// TwinCAT 3 PLC project Plc
// ProgramVersion: 3.1.4024.0
// libraries:
//   Tc2_Math, * (Beckhoff Automation GmbH)
//   Tc2_MC2, * (Beckhoff Automation GmbH)
//   Tc2_Standard, * (Beckhoff Automation GmbH)
//   Tc2_System, * (Beckhoff Automation GmbH)
//   Tc3_Module, * (Beckhoff Automation GmbH)
// project tree:
//   DUTs/ E_Aquisition_State.TcDUT, E_TestAccuracy_State.TcDUT
//   GVLs/ GVL_AccuracyTest.TcGVL, GVL_Interpolation.TcGVL
//   / PlcTask.TcTTO
//   POUs/ Accuracy_Measurement.TcPOU, MAIN.TcPOU, PositionCompensation_1D.TcPOU
//   POUs/Maths/ average.TcPOU, max_abs_array.TcPOU, max_array.TcPOU, min_array.TcPOU, scaling.TcPOU, sigma.TcPOU
// real-time tasks:
//   TASK Task_Plc: cycle T#2ms, priority 20, ADS port 350
// motion (NC):
//   TASK NC-Task 1 SAF: cycle T#2ms, priority 4, ADS port 501
//   TASK NC-Task 1 SVB: cycle T#10ms, priority 8, ADS port 511
//   AXIS Axis 1 (id 1)
//     Dynamic: Acceleration=1225.67, Deceleration=1225.67, Jerk=3677.02
//     Velo: RefSearch=8.17116, RefSync=8.17116, SlowManual=40.8558, FastManual=245.1348, Fast=817.116, Maximum=817.116
//     TargetPosControl: Range=0.0002, Time=0.1
//     OtherSettings: AllowMotionCmdToSlave=true
//     encoder EncType=19
//       EncPara: ScaleFactorNumerator=10, ScaleFactorDenominator=1048576, MaxCount=#xffffffff
//         SoftEndMinControl: Enable=true, Range=-170
//         SoftEndMaxControl: Enable=true, Range=30
//     drive DrvType=16
//       DrvPara: MaxCount=#xffffffff, DriveControlDWord=#x00020100
//         Analog: VeloReferenz=898.8276, VeloScale=71.5255737304688, TorqueSetpointScale=10, ScaleFactorActTorque=0.1
//         TimeComp: TaskDelayCycles=1
//     controller CtrType=1
//       CtrPara: PriorControlFactor=1
//         Observer: BandWidth=20
//   AXIS Axis 2 (id 2)
//     Dynamic: Acceleration=5539.8765, Deceleration=5539.8765, Jerk=16619.6295
//     Velo: RefSearch=36.93251, RefSync=36.93251, SlowManual=184.66255, FastManual=1107.9753, Fast=3693.251, Maximum=3693.251
//     TargetPosControl: Range=0.0005, Time=0.1
//     OtherSettings: AllowMotionCmdToSlave=true
//     encoder EncType=19
//       EncPara: ScaleFactorNumerator=60, ScaleFactorDenominator=1048576, MaxCount=#xffffffff
//     drive DrvType=16
//       DrvPara: MaxCount=#xffffffff, DriveControlDWord=#x00020100
//         Analog: VeloReferenz=4062.5761, VeloScale=71.5255737304688, TorqueSetpointScale=10, ScaleFactorActTorque=0.1
//         TimeComp: TaskDelayCycles=1
//     controller CtrType=1
//       CtrPara: PriorControlFactor=1
//         Observer: BandWidth=20
// I/O:
//   DEVICE Device 1 (EtherCAT) (disabled), AmsNetId 5.64.37.70.2.1
//     Term 1 (EK1200) [EK1200-5000 EtherCAT Power supply (2A E-Bus)]
//       Term 2 (EL6910) [EL6910, TwinSAFE PLC]
//       Term 3 (EL1904) [EL1904, 4 Ch. Safety Input 24V, TwinSAFE]
//         modules: Module 1 (FSOES)
//       Term 4 (EL1008) [EL1008 8Ch. Dig. Input 24V, 3ms]
//       Term 5 (EL9011) [EL9011 End Terminal]
//   DEVICE Device 4 (EtherCAT), AmsNetId 5.64.37.70.5.1
//     Term 6 (AX8620-0000-0103) [AX8620-0000-0103]
//       Drive 7 (AX8206-0210-0106) [AX8206-0210-0106 (2Ch. 6A servo axis, safe-motion, multi-FB)]
//         modules: Device, Device, Device, Device, Device, Device, Device, Device, Device, Device, Device (Safety), Device, Device, Device, Device, Device, Device, Device, Device, Device, Device, Device, Device, Device, Device, Device, Device, Device, Device, Device, Device, Ch A, Ch A, Ch A, Ch A, Ch A, Ch A, Ch A, Ch A, Ch A, Ch A, Ch A, Ch A, Ch A, Ch A, Ch A, Ch A, Ch A, Ch A, Ch A, Ch A, Ch A, Ch A, Ch A, Ch A, Ch A, Ch A, Ch A, Ch B, Ch B, Ch B, Ch B, Ch B, Ch B, Ch B, Ch B, Ch B, Ch B, Ch B, Ch B, Ch B, Ch B, Ch B, Ch B, Ch B, Ch B, Ch B, Ch B, Ch B, Ch B, Ch B, Ch B, Ch B, Ch B
//         startup 12992:1 := 414D383032312D78427830 // Ch A Motor parameters / Configured motor type
//         startup 24768:0 := FEFF // Ch A Interpolation sub mode select
//         startup 13000:5 := 0200 // Ch A Motor thermal model / Reaction
//         startup 13000:6 := 0000C841 // Ch A Motor thermal model / Partial fraction factor
//         startup 12992:12 := 0000FA45 // Ch A Motor parameters / Motor rated speed
//         startup 12992:13 := C9E5FF3E // Ch A Motor parameters / Motor rated torque
//         startup 24694:0 := F4010000 // Ch A Motor standstill torque
//         startup 24800:0 := D007 // Ch A Positive torque/force limit value
//         startup 24801:0 := D007 // Ch A Negative torque/force limit value
//         startup 12288:6 := 4158383230362D303231302D30303030 // Ch A AxisMain parameters / Configured drive type
//         startup 12867:1 := 9A99593F // Ch A TorqueCtrl parameters / Configured channel rated current
//         startup 12867:2 := 33332340 // Ch A TorqueCtrl parameters / Configured channel peak current
//         startup 12867:7 := 77BE1F40 // Ch A TorqueCtrl parameters / Iuvw max sum
//         startup 24672:0 := 08 // Ch A Modes of operation
//         startup 13023:0 := 0000 // Ch A Motor control mode
//         startup 12864:1 := 0D4D7043 // Ch A TorqueCtrl parameters mappable / Torque control proportional gain q
//         startup 12864:2 := 8A0E7C39 // Ch A TorqueCtrl parameters mappable / Torque control integral action time q
//         startup 12608:1 := FBD1CD3B // Ch A VeloCtrl parameters mappable / Velocity control proportional gain
//         startup 12608:2 := 6F12033C // Ch A VeloCtrl parameters mappable / Velocity control integral action time
//         startup 12608:3 := 00980546 // Ch A VeloCtrl parameters mappable / Bipolar velocity limit value
//         startup 12992:15 := 0100 // Ch A Motor parameters / Motor temperature sensor connection
//         startup 12611:4 := 0400 // Ch A VeloCtrl observer / Observer type
//         startup 24672:0 := 08 // Ch A Modes of operation
//         startup 12296:2 := 00 // Ch A AxisMain parameters encoder direction / Primary encoder direction
//         startup 12296:1 := 00 // Ch A AxisMain parameters encoder direction / Secondary encoder direction
//         startup 14016:1 := 414D383033332D78467831 // Ch B Motor parameters / Configured motor type
//         startup 26816:0 := FEFF // Ch B Interpolation sub mode select
//         startup 14024:5 := 0200 // Ch B Motor thermal model / Reaction
//         startup 14024:6 := 0000C841 // Ch B Motor thermal model / Partial fraction factor
//         startup 14016:12 := 0080BB45 // Ch B Motor parameters / Motor rated speed
//         startup 14016:13 := 2FDD3440 // Ch B Motor parameters / Motor rated torque
//         startup 26742:0 := 920C0000 // Ch B Motor standstill torque
//         startup 26848:0 := D007 // Ch B Positive torque/force limit value
//         startup 26849:0 := D007 // Ch B Negative torque/force limit value
//         startup 13312:6 := 4158383230362D303231302D30303030 // Ch B AxisMain parameters / Configured drive type
//         startup 13891:1 := 33338340 // Ch B TorqueCtrl parameters / Configured channel rated current
//         startup 13891:2 := CDCC4441 // Ch B TorqueCtrl parameters / Configured channel peak current
//         startup 13891:7 := 77BE1F40 // Ch B TorqueCtrl parameters / Iuvw max sum
//         startup 26720:0 := 08 // Ch B Modes of operation
//         startup 14047:0 := 0000 // Ch B Motor control mode
//         startup 13888:1 := 3DD94842 // Ch B TorqueCtrl parameters mappable / Torque control proportional gain q
//         startup 13888:2 := 8A0E7C39 // Ch B TorqueCtrl parameters mappable / Torque control integral action time q
//         startup 13632:1 := 4D288C3D // Ch B VeloCtrl parameters mappable / Velocity control proportional gain
//         startup 13632:2 := 6F12033C // Ch B VeloCtrl parameters mappable / Velocity control integral action time
//         startup 13632:3 := 00980546 // Ch B VeloCtrl parameters mappable / Bipolar velocity limit value
//         startup 14016:15 := 0100 // Ch B Motor parameters / Motor temperature sensor connection
//         startup 13635:4 := 0400 // Ch B VeloCtrl observer / Observer type
//         startup 26720:0 := 08 // Ch B Modes of operation
//         startup 13320:2 := 00 // Ch B AxisMain parameters encoder direction / Primary encoder direction
// variable links:
//   Device 4 (EtherCAT) <-> Device 4 (EtherCAT)/Term 6 (AX8620-0000-0103)/Drive 7 (AX8206-0210-0106)
//     Term 6 (AX8620-0000-0103)/PSM Controlword for axis/Controlword for axis <-> Device/DeviceMain Outputs/Power supply controlword
//   NC-Task 1 SAF/Axes/Axis 1 <-> Device 4 (EtherCAT)/Term 6 (AX8620-0000-0103)/Drive 7 (AX8206-0210-0106)
//     Drive/Inputs/In/nDataIn1 <-> Ch A/Ch A PositionControl Inputs/Ch A Following error actual value
//     Drive/Inputs/In/nDataIn3[0] <-> Ch A/Ch A TorqueControl Inputs/Ch A Torque/force actual value
//     Drive/Inputs/In/nDcOutputTime <-> InfoData/DcOutputShift
//     Drive/Inputs/In/nState1 <-> Ch A/Ch A AxisMain Inputs/Ch A Statusword
//     Drive/Inputs/In/nState2 <-> Ch A/Ch A AxisMain Inputs/Ch A Statusword @bit 8
//     Drive/Inputs/In/nState4 @bit 1 <-> WcState/InputToggle0
//     Drive/Inputs/In/nState4 <-> WcState/WcState0
//     Drive/Outputs/Out/nCtrl1 <-> Ch A/Ch A AxisMain Outputs/Ch A Controlword
//     Drive/Outputs/Out/nCtrl2 <-> Ch A/Ch A AxisMain Outputs/Ch A Controlword @bit 8
//     Drive/Outputs/Out/nDataOut1 <-> Ch A/Ch A Interpolator Outputs/Ch A Target position
//     Drive/Outputs/Out/nDataOut2 <-> Ch A/Ch A Interpolator Outputs/Ch A Target velocity
//     Enc/Inputs/In/nDataIn1 <-> Ch A/Ch A AxisMain Inputs/Ch A Position actual value
//     Enc/Inputs/In/nDcInputTime <-> InfoData/DcInputShift
//     Enc/Inputs/In/nState2 @bit 5 <-> Ch A/Ch A AxisMain Inputs/Position actual value invalid
//     Enc/Inputs/In/nState4 @bit 1 <-> WcState/InputToggle0
//     Enc/Inputs/In/nState4 <-> WcState/WcState0
//   NC-Task 1 SAF/Axes/Axis 2 <-> Device 4 (EtherCAT)/Term 6 (AX8620-0000-0103)/Drive 7 (AX8206-0210-0106)
//     Drive/Inputs/In/nDataIn1 <-> Ch B/Ch B PositionControl Inputs/Ch B Following error actual value
//     Drive/Inputs/In/nDcOutputTime <-> InfoData/DcOutputShift
//     Drive/Inputs/In/nState1 <-> Ch B/Ch B AxisMain Inputs/Ch B Statusword
//     Drive/Inputs/In/nState2 <-> Ch B/Ch B AxisMain Inputs/Ch B Statusword @bit 8
//     Drive/Inputs/In/nState4 @bit 1 <-> WcState/InputToggle0
//     Drive/Inputs/In/nState4 <-> WcState/WcState0
//     Drive/Outputs/Out/nCtrl1 <-> Ch B/Ch B AxisMain Outputs/Ch B Controlword
//     Drive/Outputs/Out/nCtrl2 <-> Ch B/Ch B AxisMain Outputs/Ch B Controlword @bit 8
//     Drive/Outputs/Out/nDataOut1 <-> Ch B/Ch B Interpolator Outputs/Ch B Target position
//     Drive/Outputs/Out/nDataOut2 <-> Ch B/Ch B Interpolator Outputs/Ch B Target velocity
//     Enc/Inputs/In/nDataIn1 <-> Ch B/Ch B AxisMain Inputs/Ch B Position actual value
//     Enc/Inputs/In/nDcInputTime <-> InfoData/DcInputShift
//     Enc/Inputs/In/nState2 @bit 5 <-> Ch B/Ch B AxisMain Inputs/Position actual value invalid
//     Enc/Inputs/In/nState4 @bit 1 <-> WcState/InputToggle0
//     Enc/Inputs/In/nState4 <-> WcState/WcState0
//   Plc/Plc Instance <-> Device 4 (EtherCAT)/Term 6 (AX8620-0000-0103)/Drive 7 (AX8206-0210-0106)
//     PlcTask Inputs/Accuracy_Measurement.iLastPositionRaw <-> Ch A/Ch A AxisMain Inputs/1st additional position actual value
//   Plc/Plc Instance <-> NC-Task 1 SAF/Axes/Axis 1
//     PlcTask Inputs/Accuracy_Measurement.Axis.NcToPlc <-> Outputs/ToPlc
//     PlcTask Outputs/Accuracy_Measurement.Axis.PlcToNc <-> Inputs/FromPlc

CONFIGURATION Plc
    RESOURCE PLC ON TwinCAT3
        TASK PlcTask(INTERVAL := T#2ms, PRIORITY := 20);
        PROGRAM MAIN WITH PlcTask : MAIN;
    END_RESOURCE
END_CONFIGURATION

// ---- DUTs/E_Aquisition_State.TcDUT
{attribute 'qualified_only'}
{attribute 'strict'}
TYPE E_Aquisition_State :
(
	IDLE := 0,
	MOVE_TO_FIRST_POS,
	WAIT_MOVE_TO_FIRST_POS,
	MOVE_TO_TARGET_FORWARD,
	WAIT_MOVE_TO_TARGET_FORWARD,
	MOVE_TO_LAST_POS,
	WAIT_MOVE_TO_LAST_POS,
	MOVE_TO_TARGET_BACKWARD,
	WAIT_MOVE_TO_TARGET_BACKWARD,
	DONE
);
END_TYPE

// ---- DUTs/E_TestAccuracy_State.TcDUT
{attribute 'qualified_only'}
{attribute 'strict'}
TYPE E_TestAccuracy_State :
(
	IDLE := 0,
	MOVE_TO_FIRST_POS,
	WAIT_MOVE_TO_FIRST_POS,
	MOVE_TO_TARGET_FORWARD,
	WAIT_MOVE_TO_TARGET_FORWARD,
	MOVE_TO_LAST_POS,
	WAIT_MOVE_TO_LAST_POS,
	MOVE_TO_TARGET_BACKWARD,
	WAIT_MOVE_TO_TARGET_BACKWARD,
	DONE
);
END_TYPE

// ---- GVLs/GVL_AccuracyTest.TcGVL
{attribute 'qualified_only'}
VAR_GLOBAL CONSTANT
	N_NBR_POSITIONS 	: UINT := 10;
	N_NBR_CYCLES 		: UINT := 5;
	N_NBR_DELAY_CYCLES 	: UINT := 5;
END_VAR

// ---- GVLs/GVL_Interpolation.TcGVL
{attribute 'qualified_only'}
VAR_GLOBAL
	N_MAX_POINTS : UINT := 10;
END_VAR

// ---- POUs/MAIN.TcPOU
PROGRAM MAIN
VAR 
END_VAR

Accuracy_Measurement();

END_PROGRAM

// ---- POUs/Accuracy_Measurement.TcPOU
PROGRAM Accuracy_Measurement
VAR
	
{region 'Axis Control FB'}	
	fbAxis 						: AXIS_REF;			// Axis to be moved
	
	fbPower						: MC_Power;			// Power the axis
	bPower						: BOOL;
	                			
	fbMove						: MC_MoveAbsolute;  // Move the axis
	bMove						: BOOL;
	fTarget						: LREAL;
	fVelocity					: LREAL := 100;
	fAcceleration				: LREAL;
	fJerk 						: LREAL;
	stOutputs					: ST_McOutputs;
		 
	fPositionError				: LREAL;			// Load Following error
	aRollingBuffer				: ARRAY[1..GVL_AccuracyTest.N_NBR_DELAY_CYCLES] OF LREAL; // Dead time of set pos
		 
	
	fbCompensation				: PositionCompensation_1D;  // Compensation
{endregion}	      	
	 
{region 'Load Position'}
	nLoadPositionRaw AT%I*		: DINT;				// Raw 
	fLoadPositionScaled 		: LREAL;			// Scaled Position in NC unit
	fLoadPositionOffset 		: LREAL := -74.157595; // To be calibrated for the current axis
{endregion}	

{region 'Cycle control'}	
	aSetposition				: ARRAY[1..GVL_AccuracyTest.N_NBR_POSITIONS] OF LREAL; // all positions for the measurement
	aMeasuredData				: ARRAY[1..GVL_AccuracyTest.N_NBR_POSITIONS, 1..2*GVL_AccuracyTest.ciNumCycles] OF LREAL; // Cycles : odd = forward, even = backward
	nCurrentSetpoint 			: UINT;			//
	nCurrentCycle	  			: UINT;
	bBackward					: BOOL;		     // Moving Backward
	fPositionMin				: LREAL := -170; // initialized from the NC
	fPositionMax				: LREAL := 30;   // initialized from the NC
	fStep						: LREAL;
{endregion}

{region 'ISO 230-2 metrics'}	
	aAverageForward					: ARRAY[1..GVL_AccuracyTest.N_NBR_POSITIONS] OF LREAL; 
	aAverageBackward				: ARRAY[1..GVL_AccuracyTest.N_NBR_POSITIONS] OF LREAL; 
	aAverageBidir					: ARRAY[1..GVL_AccuracyTest.N_NBR_POSITIONS] OF LREAL; 
	aSigmaForward					: ARRAY[1..GVL_AccuracyTest.N_NBR_POSITIONS] OF LREAL; 
	aSigmaBackward					: ARRAY[1..GVL_AccuracyTest.N_NBR_POSITIONS] OF LREAL; 
	aReversal						: ARRAY[1..GVL_AccuracyTest.N_NBR_POSITIONS] OF LREAL; 
	fReversalValue					: LREAL;
	aRepeatabilityForward 			: ARRAY[1..GVL_AccuracyTest.N_NBR_POSITIONS] OF LREAL;
	aRepeatabilityBackward 			: ARRAY[1..GVL_AccuracyTest.N_NBR_POSITIONS] OF LREAL;
	aRepeatabilityBidir				: ARRAY[1..GVL_AccuracyTest.N_NBR_POSITIONS] OF LREAL;
	fRepeatForward					: LREAL;
	fRepeatBackWard					: LREAL;
	fRepeatBidir					: LREAL;
	fSystematicAccuracyForward 		: LREAL;
	fSystematicAccuracyBackward		: LREAL;
	fSystematicAccuracyBidir 		: LREAL;
	fAverageBidirError				: LREAL;
	fAccuracyForward 				: LREAL;
	fAccuracyBackward 				: LREAL;
	fAccuracyBidir					: LREAL;	
{endregion}
	

          			

{region 'Inialization'}                			
	fScalingNum					: LREAL;
	fScalingDenum				: LREAL;
	                    		
	fbReadAccel					: MC_ReadParameter;
	fbReadJerk					: MC_ReadParameter;
	fbReadScalingNum			: MC_ReadParameter;
	fbReadScalingDenum			: MC_ReadParameter;
	fbReadMinPos				: MC_ReadParameter;
	fbReadMaxPos				: MC_ReadParameter;	 
{endregion}
	 
	
{region 'commands of the program'} 
	
	{attribute 'init_on_onlchange' }
	bInit						: BOOL;					// Start the initalization
	{attribute 'init_on_onlchange' }
	bRead						: BOOL;					// Read the init data			
	
	bStartMeasure				: BOOL;					// Start the accuracy measurement cycle
	nStateMeasure				: E_Aquisition_State;
	
	bCompute					: BOOL;					// Start the metrics computation
	
	bTestAccuracy 				: BOOL;					// Execute the cycle without measurement
	nStateTestAccuracy			: E_TestAccuracy_State;
		 
	bStop 						: BOOL;					// Stop cycles
	
	// Data for Scope Display
	fDisplaySetpointForward, fDisplaySetpointBackward, fDisplayMeasurementForward, fDisplayMeasurementBackward 	: LREAL;
	fDisplaySetpointComput, fDisplayMeasurementAverageForward, fDisplayMeasurementAverageBackward 				: LREAL;
	
	bCompensate					: BOOL;					// Start usung the compensation
{endregion}	

	

END_VAR

// Don't go further if not init
IF NOT bInit THEN
	 bRead := TRUE;
	 Init();
	 RETURN;
END_IF


//Start Acquistion
IF bStartMeasure THEN
	IF fbAxis.Status.Disabled THEN
		bPower := TRUE;
	ELSE
		nCurrentCycle := 0;
		nCurrentSetpoint := 1;
		nStateMeasure := E_Aquisition_State.MOVE_TO_FIRST_POS;
		bStartMeasure := FALSE;
	END_IF
END_IF

//Start Measurement
IF bTestAccuracy THEN
	IF fbAxis.Status.Disabled THEN
		bPower := TRUE;
	ELSE
		nCurrentSetpoint := 1;
		nStateTestAccuracy := E_TestAccuracy_State.MOVE_TO_FIRST_POS;
		bTestAccuracy := FALSE;
	END_IF
END_IF

// Compute the metrics
IF bCompute THEN
	bCompute := FALSE;
	Compute();
END_IF


// Cyclic Update
Cycle();
Acquisition();
TestAccuracy();

METHOD Acquisition : BOOL
(* This method moves the axis and aquires the position data to be processed later in the compute method *)

CASE nStateMeasure OF
	E_Aquisition_State.IDLE: // IDLE
		;
		
	E_Aquisition_State.MOVE_TO_FIRST_POS:
		fTarget := fPositionMin;
		bMove := TRUE;
		nStateMeasure := E_Aquisition_State.WAIT_MOVE_TO_FIRST_POS;
		
	E_Aquisition_State.WAIT_MOVE_TO_FIRST_POS:
		IF stOutputs.Done THEN
			bMove := FALSE;
			nStateMeasure :=  E_Aquisition_State.MOVE_TO_TARGET_FORWARD;
			nCurrentCycle	 := nCurrentCycle+1;
			nCurrentSetpoint := 1;
		END_IF
		
		IF nCurrentCycle > 2*GVL_AccuracyTest.N_NBR_CYCLES THEN
			nStateMeasure :=  E_Aquisition_State.DONE;
		END_IF
		
	E_Aquisition_State.MOVE_TO_TARGET_FORWARD:
		fTarget := aSetposition[nCurrentSetpoint];
		bMove := TRUE;
		nStateMeasure := E_Aquisition_State.WAIT_MOVE_TO_TARGET_FORWARD;
		
	E_Aquisition_State.WAIT_MOVE_TO_TARGET_FORWARD:
		IF stOutputs.Done  THEN
			bMove := FALSE;
			aMeasuredData[nCurrentSetpoint,nCurrentCycle] := fLoadPositionScaled-aSetposition[nCurrentSetpoint];
			fDisplayMeasurementForward := aMeasuredData[nCurrentSetpoint,nCurrentCycle];
			fDisplaySetpointForward := aSetposition[nCurrentSetpoint];
			nStateMeasure := E_Aquisition_State.MOVE_TO_TARGET_FORWARD;
			nCurrentSetpoint := nCurrentSetpoint+1;		
		END_IF
		IF nCurrentSetpoint > GVL_AccuracyTest.N_NBR_POSITIONS THEN
			nStateMeasure := E_Aquisition_State.MOVE_TO_LAST_POS;
		END_IF
		
	E_Aquisition_State.MOVE_TO_LAST_POS : 
		fTarget := fPositionMax;
		bMove := TRUE;
		nStateMeasure := E_Aquisition_State.WAIT_MOVE_TO_LAST_POS;	
	
	E_Aquisition_State.WAIT_MOVE_TO_LAST_POS:
		IF stOutputs.Done THEN
			bMove := FALSE;
			nStateMeasure := E_Aquisition_State.WAIT_MOVE_TO_TARGET_BACKWARD;
			nCurrentSetpoint := GVL_AccuracyTest.N_NBR_POSITIONS;
			nCurrentCycle	 := nCurrentCycle+1;
		END_IF		
		IF nCurrentCycle > 2*GVL_AccuracyTest.N_NBR_CYCLES THEN
			nStateMeasure := E_Aquisition_State.DONE;
		END_IF
		
	E_Aquisition_State.MOVE_TO_TARGET_BACKWARD:
		fTarget := aSetposition[nCurrentSetpoint];
		bMove := TRUE;
		nStateMeasure := E_Aquisition_State.WAIT_MOVE_TO_TARGET_BACKWARD;
		
	E_Aquisition_State.WAIT_MOVE_TO_TARGET_BACKWARD:
		IF stOutputs.Done  THEN
			bMove := FALSE;
			aMeasuredData[nCurrentSetpoint,nCurrentCycle] := fLoadPositionScaled-aSetposition[nCurrentSetpoint];
			fDisplayMeasurementBackward := aMeasuredData[nCurrentSetpoint,nCurrentCycle];
			fDisplaySetpointBackward := aSetposition[nCurrentSetpoint];
			nStateMeasure := E_Aquisition_State.MOVE_TO_TARGET_BACKWARD;
			nCurrentSetpoint := nCurrentSetpoint-1;		
		END_IF
		IF nCurrentSetpoint < 1 THEN
			nStateMeasure := E_Aquisition_State.MOVE_TO_FIRST_POS;
		END_IF
		
	E_Aquisition_State.DONE:
		bCompute := TRUE;
		nStateMeasure := E_Aquisition_State.IDLE;

END_CASE
END_METHOD

METHOD Compute : BOOL
VAR
	i , j : UINT;
	aTempDataForward : ARRAY[1..GVL_AccuracyTest.N_NBR_CYCLES] OF LREAL;
	aTempDataBackward : ARRAY[1..GVL_AccuracyTest.N_NBR_CYCLES] OF LREAL;
	lrMaxForward		: LREAL;
	lrMinForward		: LREAL;
	lrMaxBackward		: LREAL;
	lrMinBackward		: LREAL;
END_VAR
(* This method computes the positioning accuracy metrics according to ISO 230-2 *)

// ***** initialization ******** //
lrMinForward  := 1E300;
lrMinBackward := 1E300;
lrMaxForward := -1E300;
lrMaxBackward := -1E300;

// ***** compute data for all positions  ******** //
FOR i := 1 TO GVL_AccuracyTest.N_NBR_POSITIONS DO
	// gather all samples for each position
	FOR j := 1 TO GVL_AccuracyTest.N_NBR_CYCLES DO
		aTempDataForward[j] := aMeasuredData[i,2*j-1];
		aTempDataBackward[j] := aMeasuredData[i,2*j];
	END_FOR
	
	// compute the average at this position
	aAverageForward[i] := average(aTempDataForward);
	aAverageBackward[i] := average(aTempDataBackward);
	aAverageBidir[i] := (aAverageForward[i]+aAverageBackward[i])/2;
	
	// compute the reversal value  at this position
	aReversal[i] := aAverageForward[i]-aAverageBackward[i];
	
	// compute the standard deviation at this position
	aSigmaForward[i] := sigma(aTempDataForward,aAverageForward[i]);
	aSigmaBackward[i] := sigma(aTempDataBackward,aAverageBackward[i]);
	
	// find the extremities of each travel
	lrMaxForward	:= MAX(lrMaxForward,aAverageForward[i]+2*aSigmaForward[i] );
	lrMinForward	:= MIN(lrMinForward,aAverageForward[i]-2*aSigmaForward[i] );
	lrMaxBackward	:= MAX(lrMaxBackward,aAverageBackward[i]+2*aSigmaBackward[i] );
	lrMinBackward   := MIN(lrMinBackward,aAverageBackward[i]-2*aSigmaBackward[i] );
	
	// compute the repeatability for each value
	aRepeatabilityForward[i] := 4*aSigmaForward[i];
	aRepeatabilityBackward[i] := 4*aSigmaBackward[i];
	aRepeatabilityBidir[i] := MAX(2*aSigmaForward[i]+2*aSigmaBackward[i]+ABS(aReversal[i]),aRepeatabilityForward[i],aRepeatabilityBackward[i]);
END_FOR


// ***** compute the metrics ******** //
//  Reversal value (maximum backlash)
fReversalValue := max_abs_array(aReversal);
// Repeatability
fRepeatForward	 := max_abs_array(aRepeatabilityForward);
fRepeatBackWard := max_abs_array(aRepeatabilityBackward);
fRepeatBidir	 := max_abs_array(aRepeatabilityBidir);
// Systematic accuracy (maximal compensation)
fSystematicAccuracyForward := max_array(aAverageForward) - min_array(aAverageForward) ;
fSystematicAccuracyBackward := max_array(aAverageBackward) - min_array(aAverageBackward) ;
fSystematicAccuracyBidir := MAX(max_array(aAverageForward),max_array(aAverageBackward)) - MIN(min_array(aAverageForward),min_array(aAverageBackward));
// Average Bidirectional error 
fAverageBidirError			:= max_array(aAverageBidir) - min_array(aAverageBidir);
//Reversal value
fAccuracyForward 	:= lrMaxForward-lrMinForward;
fAccuracyBackward 	:= lrMaxBackward- lrMinBackward;
fAccuracyBidir		:= MAX(lrMaxForward,lrMaxBackward)-MIN(lrMinForward,lrMinBackward);

// ***** OPTIONAL start the compensation using this data ******** //
// xCompensate := TRUE;
END_METHOD

METHOD Cycle : BOOL
VAR
	i : DINT;
END_VAR
(* This method takes care of cyclic updates *)

// Keep the axis status up to date
fbAxis.ReadStatus();

// Manage power of the motor
fbPower(
	Axis:= fbAxis, 
	Enable:= bPower, 
	Enable_Positive:= TRUE, 
	Enable_Negative:= TRUE, 
	Override:= 100, 
	BufferMode:= , 
	Options:= , 
	Status=> , 
	Busy=> , 
	Error=> , 
	ErrorID=> );

// Manage the move absolute command
fbMove(
	Axis:= fbAxis, 
	Execute:= bMove, 
	Position:= fTarget, 
	Velocity:= fVelocity, 
	Acceleration:= fAcceleration, 
	Deceleration:= fAcceleration, 
	Jerk:= fJerk, 
	BufferMode:= , 
	Options:= , 
	Done=> stOutputs.Done, 
	Busy=> stOutputs.Busy, 
	Active=> stOutputs.Active, 
	CommandAborted=> stOutputs.CommandAborted, 
	Error=> stOutputs.Error, 
	ErrorID=> stOutputs.ErrorID);
	
// Compensate the accuracy
fbCompensation(
	afCompensationTableForward:= aAverageForward, 
	afCompensationTableBackward:= aAverageBackward, 
	fbAxis:= fbAxis, 
	fStartPosition:= aSetposition[1], 
	fStopPosition:= aSetposition[GVL_AccuracyTest.N_NBR_POSITIONS], 
	bEnable:= bCompensate);
	
//	Load position 
fLoadPositionScaled := Scaling(fInput := nLoadPositionRaw, fScalingNum := fScalingNum, fScalingDenum := fScalingDenum) + fLoadPositionOffset;

// Dead time of the Set Position computed in the PLC 
FOR i := 1 TO  3 DO
	aRollingBuffer[i] := aRollingBuffer[i+1];
END_FOR
aRollingBuffer[i] := fbAxis.NcToPlc.SetPos;

// Load following error
fPositionError := aRollingBuffer[1] - fLoadPositionScaled ;
END_METHOD

METHOD Init : BOOL
VAR
	bValid : BOOL := TRUE;
END_VAR
(* This method reads initialization data from the NC Axis directly *)

bValid := TRUE; 

// Init the acceleration value
fbReadAccel(
	Axis:= fbAxis, 
	Enable:= bRead, 
	ParameterNumber:= MC_AxisParameter.AxisAcc, 
	ReadMode:= E_ReadMode.READMODE_CYCLIC, 
	Valid=> , 
	Busy=> , 
	Error=> , 
	ErrorID=> , 
	Value=> fAcceleration);	
	bValid := bValid AND fbReadAccel.Valid;

// Init the jerk value
fbReadJerk(
	Axis:= fbAxis, 
	Enable:= bRead, 
	ParameterNumber:= MC_AxisParameter.AxisJerk, 
	ReadMode:= E_ReadMode.READMODE_CYCLIC, 
	Valid=> , 
	Busy=> , 
	Error=> , 
	ErrorID=> , 
	Value=> fJerk);	
	bValid := bValid AND fbReadJerk.Valid;
	
// Read the denominator scaling value
fbReadScalingDenum(
	Axis:= fbAxis, 
	Enable:= bRead, 
	ParameterNumber:= MC_AxisParameter.AxisEncoderScalingDenominator, 
	ReadMode:= E_ReadMode.READMODE_CYCLIC, 
	Valid=> , 
	Busy=> , 
	Error=> , 
	ErrorID=> , 
	Value=> fScalingDenum);	
	bValid := bValid AND fbReadScalingDenum.Valid;

// Read the numerator scaling value
fbReadScalingNum(
	Axis:= fbAxis, 
	Enable:= bRead, 
	ParameterNumber:= MC_AxisParameter.AxisEncoderScalingNumerator, 
	ReadMode:= E_ReadMode.READMODE_CYCLIC, 
	Valid=> , 
	Busy=> , 
	Error=> , 
	ErrorID=> , 
	Value=> fScalingNum);	
	bValid := bValid AND fbReadScalingNum.Valid;

// Read the minimum position
fbReadMinPos(
	Axis:= fbAxis, 
	Enable:= bRead, 
	ParameterNumber:= MC_AxisParameter.AxisMinSoftPosLimit , 
	ReadMode:= E_ReadMode.READMODE_CYCLIC, 
	Valid=> , 
	Busy=> , 
	Error=> , 
	ErrorID=> , 
	Value=> fPositionMin);
	bValid := bValid AND fbReadMinPos.Valid;
	
// Read the maximal position
fbReadMaxPos(
	Axis:= fbAxis, 
	Enable:= bRead, 
	ParameterNumber:= MC_AxisParameter.AxisMaxSoftPosLimit, 
	ReadMode:= E_ReadMode.READMODE_CYCLIC, 
	Valid=> , 
	Busy=> , 
	Error=> , 
	ErrorID=> , 
	Value=> fPositionMax);
	bValid := bValid AND fbReadMaxPos.Valid;

	
// If all data is valid, we initialize the steps where the data will be aquired
// NOTE : we should add a random part for the positions, in order to comply with the norm ISO 230-2	but this is not done here
IF bValid THEN
	fStep := (fPositionMax-fPositionMin)/ UINT_TO_LREAL(GVL_AccuracyTest.N_NBR_POSITIONS +1);
	FOR nCurrentSetpoint := 1 TO GVL_AccuracyTest.N_NBR_POSITIONS DO
		aSetposition[nCurrentSetpoint] := fStep*UINT_TO_LREAL(nCurrentSetpoint) + fPositionMin;
	END_FOR
	bInit := TRUE;
	bRead := FALSE;
END_IF
END_METHOD

METHOD TestAccuracy : BOOL
(* This method moves the axis without aquiring the position data *)

CASE nStateTestAccuracy OF
	
	E_TestAccuracy_State.IDLE: // IDLE
		;
		
	E_TestAccuracy_State.MOVE_TO_FIRST_POS:
		fTarget := fPositionMin;
		bMove := TRUE;
		nStateTestAccuracy := E_TestAccuracy_State.WAIT_MOVE_TO_FIRST_POS;
		
	E_TestAccuracy_State.WAIT_MOVE_TO_FIRST_POS:
		IF stOutputs.Done THEN						
			bMove := FALSE;
			nStateTestAccuracy := E_TestAccuracy_State.MOVE_TO_TARGET_FORWARD;
			nCurrentSetpoint := 1;
		END_IF
		
		IF bStop THEN 
			nStateTestAccuracy := E_TestAccuracy_State.DONE;
		END_IF
		
	E_TestAccuracy_State.MOVE_TO_TARGET_FORWARD:
		fTarget := aSetposition[nCurrentSetpoint];
		bMove := TRUE;
		nStateTestAccuracy := E_TestAccuracy_State.WAIT_MOVE_TO_TARGET_FORWARD;
		
	E_TestAccuracy_State.WAIT_MOVE_TO_TARGET_FORWARD:
		IF stOutputs.Done  THEN
			bMove := FALSE;
			nStateTestAccuracy := E_TestAccuracy_State.MOVE_TO_TARGET_FORWARD;
			nCurrentSetpoint := nCurrentSetpoint+1;		
		END_IF
		IF nCurrentSetpoint > GVL_AccuracyTest.N_NBR_POSITIONS THEN
			nStateTestAccuracy := E_TestAccuracy_State.MOVE_TO_LAST_POS;
		END_IF
		
	E_TestAccuracy_State.MOVE_TO_LAST_POS : 
		fTarget := fPositionMax;
		bMove := TRUE;
		nStateTestAccuracy := E_TestAccuracy_State.WAIT_MOVE_TO_LAST_POS;	
	
	E_TestAccuracy_State.WAIT_MOVE_TO_LAST_POS:
		IF stOutputs.Done THEN
			bMove := FALSE;
			nStateTestAccuracy := E_TestAccuracy_State.MOVE_TO_TARGET_BACKWARD;
			nCurrentSetpoint := GVL_AccuracyTest.N_NBR_POSITIONS;
		END_IF		
		IF bStop THEN
			nStateTestAccuracy := E_TestAccuracy_State.DONE;
		END_IF
		
	E_TestAccuracy_State.MOVE_TO_TARGET_BACKWARD:
		fTarget := aSetposition[nCurrentSetpoint];
		bMove := TRUE;
		nStateTestAccuracy := E_TestAccuracy_State.WAIT_MOVE_TO_TARGET_BACKWARD;
		
	E_TestAccuracy_State.WAIT_MOVE_TO_TARGET_BACKWARD:
		IF stOutputs.Done  THEN
			bMove := FALSE;
			nStateTestAccuracy := E_TestAccuracy_State.MOVE_TO_TARGET_BACKWARD;
			nCurrentSetpoint := nCurrentSetpoint-1;		
		END_IF
		IF nCurrentSetpoint < 1 THEN
			nStateTestAccuracy := E_TestAccuracy_State.MOVE_TO_FIRST_POS;
		END_IF
		
	E_TestAccuracy_State.DONE:
		nStateTestAccuracy := E_TestAccuracy_State.IDLE;

END_CASE
END_METHOD

END_PROGRAM

// ---- POUs/PositionCompensation_1D.TcPOU
FUNCTION_BLOCK PositionCompensation_1D
VAR_IN_OUT
	afCompensationTableForward 	: ARRAY[*] OF LREAL;	 // Compensation table (measured differences between actual pos and set pos) in NC unit
	afCompensationTableBackward : ARRAY[*] OF LREAL;	 // Compensation table (measured differences between actual pos and set pos) in NC unit
END_VAR
VAR_INPUT
	fbAxis											: REFERENCE TO AXIS_REF;	// NC axis to be compensated
	fStartPosition									: LREAL;					// First position where compensation is used in NC unit
	fStopPosition									: LREAL;					// Last position where compensation is used in NC unit
	bEnable											: BOOL;						// TRUE : position is compensated, FALSE : position is not compensated 
	fBacklashValue									: LREAL		:= 0;			// Backlash value to compensate when moving backwards in NC unit 
	fSpeedThresholdForMovementDirectionDetection	: LREAL := 0.05	;			// Threshold to detect a movement direction based on the speed in NC unit
END_VAR
VAR
	bInitDone			: BOOL := FALSE;
	nActualNbPoints		: UINT;									// How many points of the table are actually used including start and stop positions
	fActualPos 			: LREAL;
	fRemainder 			: LREAL;
	nCurrentIndex 		: UINT;
	fIndex				: LREAL;
	fCorrectionValue 	: LREAL;
	bMovingForward		: BOOL;
	fCorrectionBacklash : LREAL	:= 0;
	fbPosCorrection 	: MC_PositionCorrectionLimiter;
	fbReadParam			: MC_ReadParameter;
	fbWriteParam		: MC_WriteBoolParameter;
	fMaxAcceleration 	: LREAL;
END_VAR

// Use the rest of the code only if Enable is on
IF NOT bEnable THEN
	RETURN;
END_IF

// Check input validity 
IF NOT CheckInputsAreValid() THEN
	RETURN;
END_IF 

// Check if initialization must be done
IF NOT bInitDone THEN
	Init();
END_IF

// Compute the position correction
ComputeCorrection();
ComputeBacklash();

fbAxis.ReadStatus();

// Assign the corrections to the NC axis
fbPosCorrection(
	Axis:= fbAxis, 
	Enable:= TRUE, 
	PositionCorrectionValue:= fCorrectionValue + fCorrectionBacklash, 
	CorrectionMode:= E_AxisPositionCorrectionMode.POSITIONCORRECTION_MODE_FAST, 
	Acceleration:= fMaxAcceleration);

METHOD CheckInputsAreValid : BOOL
(* This method returns true if the inputs are valid *)
CheckInputsAreValid := FALSE;

IF  LOWER_BOUND(afCompensationTableForward,1) = LOWER_BOUND(afCompensationTableBackward,1) // check tables correspond
	AND_THEN UPPER_BOUND(afCompensationTableForward,1) = UPPER_BOUND(afCompensationTableBackward,1)
	AND fStartPosition < fStopPosition	// Make sure the direction of the points is positive	
	AND __ISVALIDREF(fbAxis) // Reference to the NC axis is valid
	THEN
		CheckInputsAreValid := TRUE;
END_IF
END_METHOD

METHOD ComputeBacklash : BOOL
(* Correct the backlash depending on the movement direction *)
IF ABS(fbAxis.NcToPlc.ActVelo) > fSpeedThresholdForMovementDirectionDetection THEN // avoid toggling at standstill
	IF fbAxis.NcToPlc.ActVelo < 0 THEN					// compensate if the movement is backward
		fCorrectionBacklash := fBacklashValue;
		bMovingForward	:= FALSE;
	ELSE
		fCorrectionBacklash := 0;
		bMovingForward	:= TRUE;
	END_IF
END_IF
END_METHOD

METHOD ComputeCorrection : BOOL
(* Reset the flag *)
ComputeCorrection := FALSE;

(* Correction of the axis based on the table (linear interpolation) *)
fActualPos := fbAxis.NcToPlc.SetPos; // get the current position
IF fActualPos > fStartPosition AND fActualPos < fStopPosition THEN // make sure we are inside the boundaries
	
	fIndex := 1 + (((fActualPos-fStartPosition)/(fStopPosition-fStartPosition)) * (nActualNbPoints-1));	// Index with fraction
	fRemainder := FRAC(fIndex);						// normalized distance from last index
	nCurrentIndex := LREAL_TO_UINT(FLOOR(fIndex));	// current table index
	
	// compute the correction value and add it to the full correction
	IF bMovingForward THEN
		fCorrectionValue := (afCompensationTableForward[nCurrentIndex+1] - afCompensationTableForward[nCurrentIndex]) * fRemainder + afCompensationTableForward[nCurrentIndex] ;
	ELSE
		fCorrectionValue := (afCompensationTableBackward[nCurrentIndex+1] - afCompensationTableBackward[nCurrentIndex]) * fRemainder + afCompensationTableBackward[nCurrentIndex] ;
	END_IF
END_IF


// Computation is done
ComputeCorrection := TRUE;
END_METHOD

METHOD PRIVATE Init : BOOL

// Read the maximum acceleration in the axis parameters
fbReadParam(
	Axis:= fbAxis, 
	Enable:= TRUE, 
	ParameterNumber:= MC_AxisParameter.AxisMaximumAcceleration, 
	ReadMode:= E_ReadMode.READMODE_ONCE, 
	Valid=> , 
	Busy=> , 
	Error=> , 
	ErrorID=> , 
	Value=> fMaxAcceleration);

// Make sure the "Enable Position Correction" parameter is TRUE	
fbWriteParam(
	Axis:= fbAxis, 
	Execute:= TRUE, 
	ParameterNumber:= MC_AxisParameter.AxisEnablePosCorrection, 
	Value:= TRUE, 
	Done=> , 
	Busy=> , 
	Error=> , 
	ErrorID=> );
	
//Get the array size
nActualNbPoints := DINT_TO_UINT(UPPER_BOUND(afCompensationTableForward,1) - LOWER_BOUND(afCompensationTableForward,1))+1;

//  If successfully intialized, set flag to true
IF fbWriteParam.Done AND NOT fbReadParam.Busy THEN
	bInitDone := TRUE;
END_IF
END_METHOD

END_FUNCTION_BLOCK

// ---- POUs/Maths/average.TcPOU
FUNCTION average : LREAL
VAR_IN_OUT
	aData : ARRAY[*] OF LREAL;
END_VAR
VAR
	nIdx  : DINT;
	fAmount, fSum : LREAL;
END_VAR

fAmount := 0;
FOR nIdx := LOWER_BOUND(aData,1) TO UPPER_BOUND(aData,1) DO
	fAmount := fAmount + 1;
    fSum := fSum + aData[nIdx] ;
END_FOR

average := fSum / fAmount;

END_FUNCTION

// ---- POUs/Maths/sigma.TcPOU
FUNCTION sigma : LREAL
VAR_IN_OUT
	aData : ARRAY[*] OF LREAL;
END_VAR
VAR_INPUT
	fAverage : LREAL;
END_VAR
VAR
	nIdx  : DINT;
	fAmount, fSum : LREAL;
END_VAR

fAmount := 0;
FOR nIdx := LOWER_BOUND(aData,1) TO UPPER_BOUND(aData,1) DO
	fAmount := fAmount + 1;
    fSum := fSum + (aData[nIdx] -fAverage)*(aData[nIdx] -fAverage) ;
END_FOR

IF fAmount > 1 THEN
	sigma := SQRT( fSum / ( fAmount-1) );
END_IF

END_FUNCTION

// ---- POUs/Maths/max_abs_array.TcPOU
FUNCTION max_abs_array : LREAL
VAR_IN_OUT
	aData : ARRAY[*] OF LREAL;
END_VAR
VAR
	nIdx: DINT;
END_VAR

max_abs_array := 0;
FOR nIdx := LOWER_BOUND(aData,1) TO UPPER_BOUND(aData,1) DO
	max_abs_array := MAX(ABS(aData[nIdx]),max_abs_array);
END_FOR

END_FUNCTION

// ---- POUs/Maths/max_array.TcPOU
FUNCTION max_array : LREAL
VAR_IN_OUT
	aData : ARRAY[*] OF LREAL;
END_VAR
VAR
	nIdx: DINT;
END_VAR

max_array := -1.7976931348623158E+308;
FOR nIdx := LOWER_BOUND(aData,1) TO UPPER_BOUND(aData,1) DO
	max_array := MAX(aData[nIdx],max_array);
END_FOR

END_FUNCTION

// ---- POUs/Maths/min_array.TcPOU
FUNCTION min_array : LREAL
VAR_IN_OUT
	aData : ARRAY[*] OF LREAL;
END_VAR
VAR
	nIdx: DINT;
END_VAR

min_array := 1.7976931348623158E+308;
FOR nIdx := LOWER_BOUND(aData,1) TO UPPER_BOUND(aData,1) DO
	min_array := MIN(aData[nIdx],min_array);
END_FOR

END_FUNCTION

// ---- POUs/Maths/scaling.TcPOU
FUNCTION scaling : LREAL
VAR_INPUT
	fInput : LREAL;
	fScalingNum : LREAL;
	fScalingDenum : LREAL;
END_VAR

Scaling := fInput * (fScalingNum / fScalingDenum);

END_FUNCTION
